// TIA Portal V18 export
// export: Created 2026-03-12T16:14:10.4682392Z, ExportSetting WithDefaults, DisplayName Totally Integrated Automation Portal, DisplayVersion V18 Update 5, DisplayName TIA Portal Openness, DisplayVersion V18 Update 5, DisplayName TIA Portal Version Control Interface, DisplayVersion V18, DisplayName SINAMICS Startdrive Advanced, DisplayVersion V18, DisplayName SINAMICS Startdrive G130, G150, S120, S150, SINAMICS MV, S210, DisplayVersion V18, DisplayName SINAMICS Startdrive G110M, G120, G120C, G120D, G120P, G115D, DisplayVersion V18, DisplayName STEP 7 Professional, DisplayVersion V18 Update 5, DisplayName STEP 7 Safety, DisplayVersion V18, DisplayName WinCC Professional, DisplayVersion V18 Update 5
Screen "TEST"  1280x800, Number=2, Template=Template Geral
  ScreenLayer 
    Group "Group"
      Rectangle "Rectang" at 320,120 size 640x130
      TextField "Text" at 360,137 size 560x96  Text="PLAYGROUND JARVIS"
    Button "Button_2" at 525,278 size 230x52  Mode=Text, Authorization=Operate, TextOff="REABRIR PLAYGROUND", TextOn="PLAYGROUND"
      on Press: ActivateScreen(Screen name := , Object number := 0)
    GraphicIOField "Graphic I/O field_15" at 580,370 size 120x120  Mode=Output, OnValue=1, PictureList=Chave seletora_1
